// TwinCAT 3 PLC project KinSimpleSample
// Title: ITcNcTrafo SampleProject
// Company: Beckhoff Automation GmbH & Co. KG
// ProgramVersion: 3.1.4023.0
// libraries:
//   Tc2_MC2, * (Beckhoff Automation GmbH)
//   Tc2_NcKinematicTransformation, * (Beckhoff Automation GmbH)
//   Tc2_Standard, * (Beckhoff Automation GmbH)
//   Tc2_System, * (Beckhoff Automation GmbH)
//   Tc3_Module, * (Beckhoff Automation GmbH)
// project tree:
//   / PlcTask.TcTTO
//   POUs/ FB_Power.TcPOU, MAIN.TcPOU
// real-time tasks:
//   TASK PlcTask: cycle T#10ms, priority 20, ADS port 350
// motion (NC):
//   TASK NC-Task 1 SAF: cycle T#2ms, priority 4, ADS port 501
//   TASK NC-Task 1 SVB: cycle T#10ms, priority 8, ADS port 511
//   AXIS J1 (id 1)
//     OtherSettings: AllowMotionCmdToSlave=true
//     encoder EncType=1
//     drive DrvType=5
//       Analog: TorqueScale=10
//       TimeComp: TaskDelayCycles=1
//     controller CtrType=1
//       CtrPara: PriorControlFactor=1
//         Observer: BandWidth=20
//   AXIS J2 (id 2)
//     OtherSettings: AllowMotionCmdToSlave=true
//     encoder EncType=1
//     drive DrvType=5
//       Analog: TorqueScale=10
//       TimeComp: TaskDelayCycles=1
//     controller CtrType=1
//       CtrPara: PriorControlFactor=1
//         Observer: BandWidth=20
//   AXIS J3 (id 3)
//     OtherSettings: AllowMotionCmdToSlave=true
//     encoder EncType=1
//     drive DrvType=5
//       Analog: TorqueScale=10
//       TimeComp: TaskDelayCycles=1
//     controller CtrType=1
//       CtrPara: PriorControlFactor=1
//         Observer: BandWidth=20
//   AXIS X (id 4)
//     OtherSettings: AllowMotionCmdToSlave=true
//     encoder EncType=1
//     drive DrvType=5
//       Analog: TorqueScale=10
//       TimeComp: TaskDelayCycles=1
//     controller CtrType=1
//       CtrPara: PriorControlFactor=1
//         Observer: BandWidth=20
//   AXIS Y (id 5)
//     OtherSettings: AllowMotionCmdToSlave=true
//     encoder EncType=1
//     drive DrvType=5
//       Analog: TorqueScale=10
//       TimeComp: TaskDelayCycles=1
//     controller CtrType=1
//       CtrPara: PriorControlFactor=1
//         Observer: BandWidth=20
//   AXIS Z (id 6)
//     OtherSettings: AllowMotionCmdToSlave=true
//     encoder EncType=1
//     drive DrvType=5
//       Analog: TorqueScale=10
//       TimeComp: TaskDelayCycles=1
//     controller CtrType=1
//       CtrPara: PriorControlFactor=1
//         Observer: BandWidth=20
// variable links:
//   KinSimpleSample/KinSimpleSample Instance <-> NC-Task 1 SAF/Axes/J1
//     PlcTask Inputs/MAIN.AxisAcs[1].NcToPlc <-> Outputs/ToPlc
//     PlcTask Outputs/MAIN.AxisAcs[1].PlcToNc <-> Inputs/FromPlc
//   KinSimpleSample/KinSimpleSample Instance <-> NC-Task 1 SAF/Axes/J2
//     PlcTask Inputs/MAIN.AxisAcs[2].NcToPlc <-> Outputs/ToPlc
//     PlcTask Outputs/MAIN.AxisAcs[2].PlcToNc <-> Inputs/FromPlc
//   KinSimpleSample/KinSimpleSample Instance <-> NC-Task 1 SAF/Axes/J3
//     PlcTask Inputs/MAIN.AxisAcs[3].NcToPlc <-> Outputs/ToPlc
//     PlcTask Outputs/MAIN.AxisAcs[3].PlcToNc <-> Inputs/FromPlc
//   KinSimpleSample/KinSimpleSample Instance <-> NC-Task 1 SAF/Axes/X
//     PlcTask Inputs/MAIN.AxisMcs[1].NcToPlc <-> Outputs/ToPlc
//     PlcTask Outputs/MAIN.AxisMcs[1].PlcToNc <-> Inputs/FromPlc
//   KinSimpleSample/KinSimpleSample Instance <-> NC-Task 1 SAF/Axes/Y
//     PlcTask Inputs/MAIN.AxisMcs[2].NcToPlc <-> Outputs/ToPlc
//     PlcTask Outputs/MAIN.AxisMcs[2].PlcToNc <-> Inputs/FromPlc
//   KinSimpleSample/KinSimpleSample Instance <-> NC-Task 1 SAF/Axes/Z
//     PlcTask Inputs/MAIN.AxisMcs[3].NcToPlc <-> Outputs/ToPlc
//     PlcTask Outputs/MAIN.AxisMcs[3].PlcToNc <-> Inputs/FromPlc
//   KinSimpleSample/KinSimpleSample Instance <-> NC-Task 1 SAF/Kin Channel
//     PlcTask Inputs/MAIN.stKinRefIn <-> Outputs/ToPlc
//     PlcTask Outputs/MAIN.stKinRefOut <-> Inputs/FromPlc

CONFIGURATION KinSimpleSample
    RESOURCE PLC ON TwinCAT3
        TASK PlcTask(INTERVAL := T#10ms, PRIORITY := 20);
        PROGRAM MAIN WITH PlcTask : MAIN;
    END_RESOURCE
END_CONFIGURATION

// ---- POUs/MAIN.TcPOU
PROGRAM MAIN
VAR
	bUserCartesianMode		: BOOL	:= TRUE;
	bUserResetKinGroup		: BOOL	:= FALSE;		
	
	AxisAcs					: ARRAY[1..3] OF AXIS_REF;
	AxisMcs					: ARRAY[1..3] OF AXIS_REF;
	
	stKinRefIn    AT %I*	: NCTOPLC_NCICHANNEL_REF;
	stKinRefOut   AT %Q*  	: PLCTONC_NCICHANNEL_REF;
		
	fbPower					: FB_Power;
	fbKinConfigGroup      	: FB_KinConfigGroup;	
	fbResetKinGroup			: FB_KinResetGroup;
	stAxesList          	: ST_KinAxes;
		
	nState					: INT := 1;
	
	bExecuteKin: BOOL;
	bKinEnableTimer : TON;
END_VAR

AxisAcs[1]();
AxisAcs[2]();
AxisAcs[3]();

AxisMcs[1]();
AxisMcs[2]();
AxisMcs[3]();

stAxesList.nAxisIdsAcs[1] := AxisAcs[1].NcToPlc.AxisId;
stAxesList.nAxisIdsAcs[2] := AxisAcs[2].NcToPlc.AxisId;
stAxesList.nAxisIdsAcs[3] := AxisAcs[3].NcToPlc.AxisId;

stAxesList.nAxisIdsMcs[1] := AxisMcs[1].NcToPlc.AxisId;
stAxesList.nAxisIdsMcs[2] := AxisMcs[2].NcToPlc.AxisId;
stAxesList.nAxisIdsMcs[3] := AxisMcs[3].NcToPlc.AxisId;


fbPower(
	bEnable :=TRUE, 
	fOvr := 100.0, 
	AxisAcs := AxisAcs,
	AxisMcs := AxisMcs, 
	bAllAxesReady=> );

CASE nState OF
	
	1:
		IF fbPower.bAllAxesReady THEN
			nState := 2;
		END_IF		
		
	2:	// The other block not coded by me takes a few more cycles to complete
		bKinEnableTimer(IN:= TRUE, PT:= T#50MS, Q=> bExecuteKin);
		IF fbKinConfigGroup.bDone THEN
			fbKinConfigGroup.bExecute := FALSE;
			nState := 3;
		END_IF
		
	3: ; //Do anything here. Build an interpolation group / move axes by hand / ...
		
END_CASE

// Configure axes according to the kinematic transformation
fbKinConfigGroup(
	bExecute:= bExecuteKin, 
	bCartesianMode:= bUserCartesianMode, 
	stAxesList:= stAxesList, 
	stKinRefIn:= stKinRefIn, 
	bBusy=> , 
	bDone=> , 
	bError=> , 
	nErrorId=> );
	
// Reset the kinematic group	
fbResetKinGroup(
	bExecute:=bUserResetKinGroup, 
	nItpChannelId:=0 , 
	stKinRefIn:= stKinRefIn, 
	stAxesList:= stAxesList, 
	bBusy=> , 
	bDone=> , 
	bError=> , 
	nErrorId=> );

END_PROGRAM

// ---- POUs/FB_Power.TcPOU
FUNCTION_BLOCK FB_Power
VAR_INPUT
	bEnable			: BOOL := FALSE;
	fOvr			: LREAL;
END_VAR
VAR_IN_OUT
	AxisAcs			: ARRAY[1..3] OF AXIS_REF;
	AxisMcs			: ARRAY[1..3] OF AXIS_REF;
END_VAR
VAR_OUTPUT
	bAllAxesReady	: BOOL := FALSE;
END_VAR
VAR
	fbPowerX		:	MC_Power;
	fbPowerY		:	MC_Power;
	fbPowerZ		:	MC_Power;
	
	fbPowerJ1		:	MC_Power;
	fbPowerJ2		:	MC_Power;
	fbPowerJ3		:	MC_Power;
END_VAR

fbPowerJ1(
	Axis:=AxisAcs[1], 
	Enable:=bEnable , 
	Enable_Positive:= bEnable, 
	Enable_Negative:= bEnable, 
	Override:=fOvr , 
	BufferMode:= , 
	Status=> , 
	Busy=> , 
	Active=> , 
	Error=> , 
	ErrorID=> );
fbPowerJ2(
	Axis:=AxisAcs[2], 
	Enable:=bEnable , 
	Enable_Positive:= bEnable, 
	Enable_Negative:= bEnable, 
	Override:=fOvr , 
	BufferMode:= , 
	Status=> , 
	Busy=> , 
	Active=> , 
	Error=> , 
	ErrorID=> );
fbPowerJ3(
	Axis:=AxisAcs[3],  
	Enable:=bEnable , 
	Enable_Positive:= bEnable, 
	Enable_Negative:= bEnable, 
	Override:=fOvr , 
	BufferMode:= , 
	Status=> , 
	Busy=> , 
	Active=> , 
	Error=> , 
	ErrorID=> );	
	
fbPowerX(
	Axis:=AxisMcs[1], 
	Enable:=bEnable , 
	Enable_Positive:= bEnable, 
	Enable_Negative:= bEnable, 
	Override:=fOvr , 
	BufferMode:= , 
	Status=> , 
	Busy=> , 
	Active=> , 
	Error=> , 
	ErrorID=> );
	
fbPowerY(
	Axis:=AxisMcs[2], 
	Enable:=bEnable , 
	Enable_Positive:= bEnable, 
	Enable_Negative:= bEnable, 
	Override:=fOvr , 
	BufferMode:= , 
	Status=> , 
	Busy=> , 
	Active=> , 
	Error=> , 
	ErrorID=> );
	
fbPowerZ(
	Axis:=AxisMcs[3],  
	Enable:=bEnable , 
	Enable_Positive:= bEnable, 
	Enable_Negative:= bEnable, 
	Override:=fOvr , 
	BufferMode:= , 
	Status=> , 
	Busy=> , 
	Active=> , 
	Error=> , 
	ErrorID=> );	
	
IF fbPowerJ1.Status AND fbPowerJ2.Status AND fbPowerJ3.Status AND fbPowerX.Status AND fbPowerY.Status AND fbPowerZ.Status THEN
	bAllAxesReady	:= TRUE;
ELSE
	bAllAxesReady	:= FALSE;
END_IF

END_FUNCTION_BLOCK
